FUNCTION_BLOCK DC_PID_FB
VAR_INPUT
	BOOL_LOW_FLOW_EN : BOOL;
	INT_HIGH_FLOW_LPM : INT;
	INT_LOW_FLOW_LPM : INT;
	INT_H_L_FLOW_RATIO : INT;
	INT_D1_LPM : INT;
	INT_D2_LPM : INT;
	INT_D3_LPM : INT;
	INT_D4_RAW : INT;
	INT_D5_RAW : INT;
	INT_D6_RAW : INT;
	INT_D1_RATIO : INT;
	INT_D2_RATIO : INT;
	INT_D3_RATIO : INT;
	INT_D4_RATIO : INT;
	INT_D5_RATIO : INT;
	INT_D6_RATIO : INT;

END_VAR

VAR_OUTPUT

	PID_FLOW_RAW : INT;
	D1_RAW_INT : INT;
	D2_RAW_INT : INT;
	D3_RAW_INT : INT;
	D4_LPM_INT : INT;
	D5_LPM_INT : INT;
	D6_LPM_INT : INT;

END_VAR
VAR
	D5EN: BOOL;
	D4EN: BOOL;
	D6EN: BOOL;
	D4REN: BOOL;
	D5REN: BOOL;
	D6REN: BOOL;
END_VAR

(*

Thats 2 program in one function block

1st Program:- 
- Let user able to select High/low flow by trigger bit "BOOL_LOW_FLOW_EN"

	Sequence detail: 
	-If "BOOL_LOW_FLOW_EN" OFF, "INT_HIGH_FLOW_LPM" will MULTIPLY "INT_H_L_FLOW_RATIO" then Feed into "PID_FLOW_RAW".
	-If "BOOL_LOW_FLOW_EN" ON, "INT_LOW_FLOW_LPM" will MULTIPLY "INT_H_L_FLOW_RATIO" then Feed into "PID_FLOW_RAW".
	-"PID_FLOW_RAW should connect direct to ANALOG OUTPUT CARD CHANNEL.


2nd Program:-
-Become Converter. Able to convert 3 types of LPM reading to RAW reading by MULTIPLY the preset RATIO.
-Become Converter. Able to convert 3 types of RAW reading to LPM reading by DIVIDE the preset RATIO.

	Sequence detail:
	-Once detected INT_D1_LPM have value (Not "0") and INT_D1_RATIO have value (Not "0") -> Program will enable and MULTIPLY "INT_D1_LPM" with "INT_D1_RATIO" and feed to "D1_RAW_INT"
	-INT_D2_LPM, INT_D2_RATIO and D2_RAW_INT function same as above (D1)
	-INT_D3_LPM, INT_D3_RATIO and D3_RAW_INT function same as above (D1)
	-Once detected INT_D4_RAW have value (Not "0") and INT_D4_RATIO have value (Not "0") -> Program will enable and DIVIDE "INT_D4_RAW" with "INT_D4_RATIO" and feed to "D4_LPM_INT"
	-INT_D5_RAW, INT_D5_RATIO and D5_LPM_INT function same as above (D4)
	-INT_D6_RAW, INT_D6_RATIO and D6_LPM_INT function same as above (D4)

*)
VAR // added by the converter: edge detectors and wires of the graphical bodies
    _w1, _w2, _w3, _w4, _w5 : INT;
END_VAR

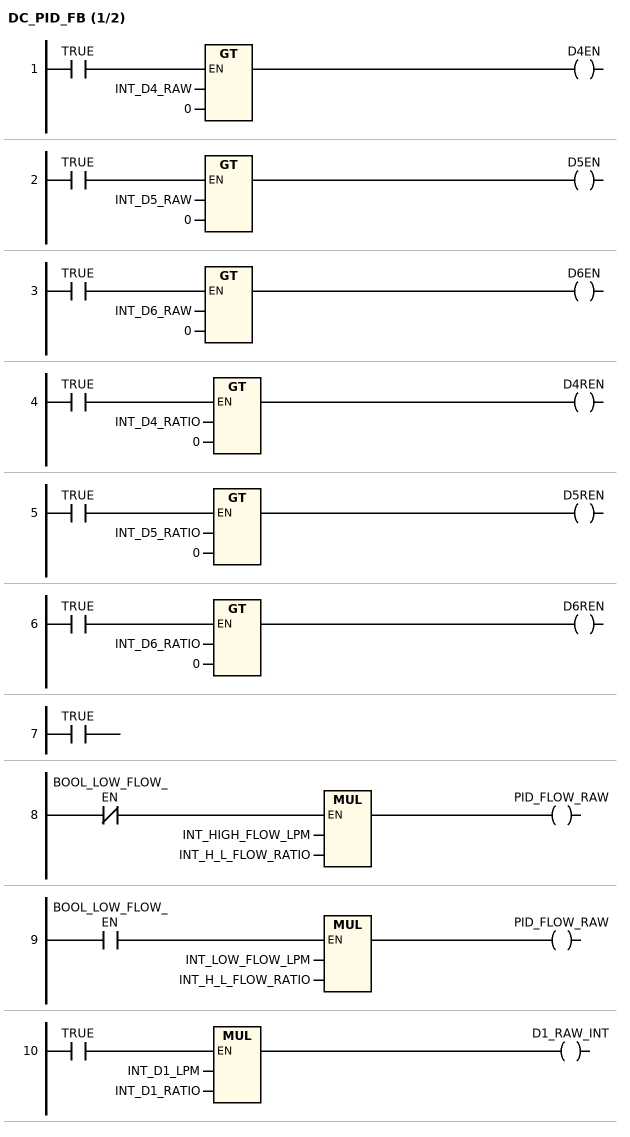
// NETWORK 1
D4EN := INT_D4_RAW > 0;

// NETWORK 2
D5EN := INT_D5_RAW > 0;

// NETWORK 3
D6EN := INT_D6_RAW > 0;

// NETWORK 4
D4REN := INT_D4_RATIO > 0;

// NETWORK 5
D5REN := INT_D5_RATIO > 0;

// NETWORK 6
D6REN := INT_D6_RATIO > 0;

// NETWORK 7

// NETWORK 8
IF NOT BOOL_LOW_FLOW_EN THEN _w1 := INT_HIGH_FLOW_LPM * INT_H_L_FLOW_RATIO; END_IF
PID_FLOW_RAW := _w1;

// NETWORK 9
IF BOOL_LOW_FLOW_EN THEN _w2 := INT_LOW_FLOW_LPM * INT_H_L_FLOW_RATIO; END_IF
PID_FLOW_RAW := _w2;

// NETWORK 10
D1_RAW_INT := INT_D1_LPM * INT_D1_RATIO;

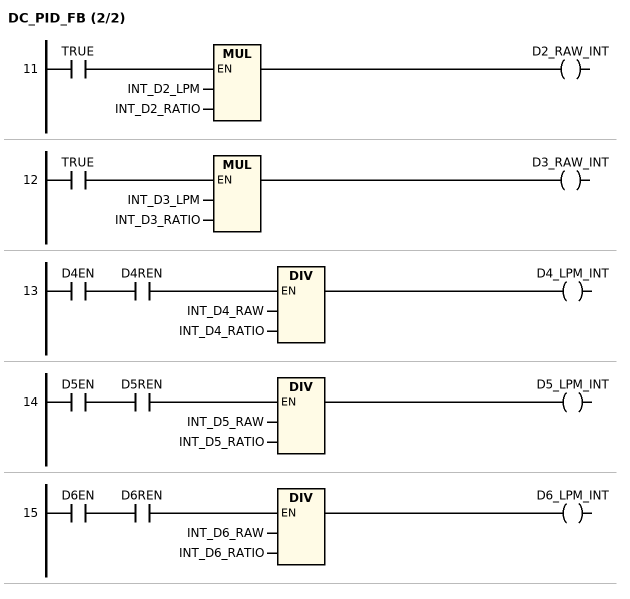
// NETWORK 11
D2_RAW_INT := INT_D2_LPM * INT_D2_RATIO;

// NETWORK 12
D3_RAW_INT := INT_D3_LPM * INT_D3_RATIO;

// NETWORK 13
IF D4EN AND D4REN THEN _w3 := INT_D4_RAW / INT_D4_RATIO; END_IF
D4_LPM_INT := _w3;

// NETWORK 14
IF D5EN AND D5REN THEN _w4 := INT_D5_RAW / INT_D5_RATIO; END_IF
D5_LPM_INT := _w4;

// NETWORK 15
IF D6EN AND D6REN THEN _w5 := INT_D6_RAW / INT_D6_RATIO; END_IF
D6_LPM_INT := _w5;

END_FUNCTION_BLOCK

(* stored: Version 1.1.0.1, ProductVersion 3.1.4024.12
   POU DC_PID_FB: Id {1ef19967-8b41-4a96-9823-cf0dcf3e7eb6}, SpecialFunc None *)
